// TIA Portal V17 export
// export: Created 2024-08-29T18:23:42.6624587Z, ExportSetting WithDefaults, DisplayName Totally Integrated Automation Portal, DisplayVersion V17 Update 7, DisplayName TIA Portal Openness, DisplayVersion V17 Update 7, DisplayName TIA Portal Version Control Interface, DisplayVersion V17, DisplayName SINAMICS Startdrive Advanced, DisplayVersion V17 SP2, DisplayName SINAMICS Startdrive G110M, G120, G120C, G120D, G120P, G115D, DisplayVersion V17 SP2, DisplayName SINAMICS Startdrive G130, G150, S120, S150, SINAMICS MV, S210, DisplayVersion V17 SP2, DisplayName STEP 7 Professional, DisplayVersion V17 Update 7, DisplayName STEP 7 Safety, DisplayVersion V17 Update 6, DisplayName WinCC Advanced / Unified PC, DisplayVersion V17 Update 7
ORGANIZATION_BLOCK "stationOutputs"   // OB124, LAD, ProgramCycle
TITLE = "Main Program Sweep (Cycle)"
{ S7_Optimized_Access := 'TRUE' }
VERSION : 0.1
// stored: AutoNumber true, IsIECCheckEnabled false, SetENOAutomatically false
   VAR_INPUT
      Initial_Call : Bool;   // Initial call of this OB
      Remanence : Bool;   // =True, if remanent data are available
   END_VAR
   VAR_TEMP
      estopOK : Bool;
   END_VAR
BEGIN

REGION Network 1: PRESENT PARTS
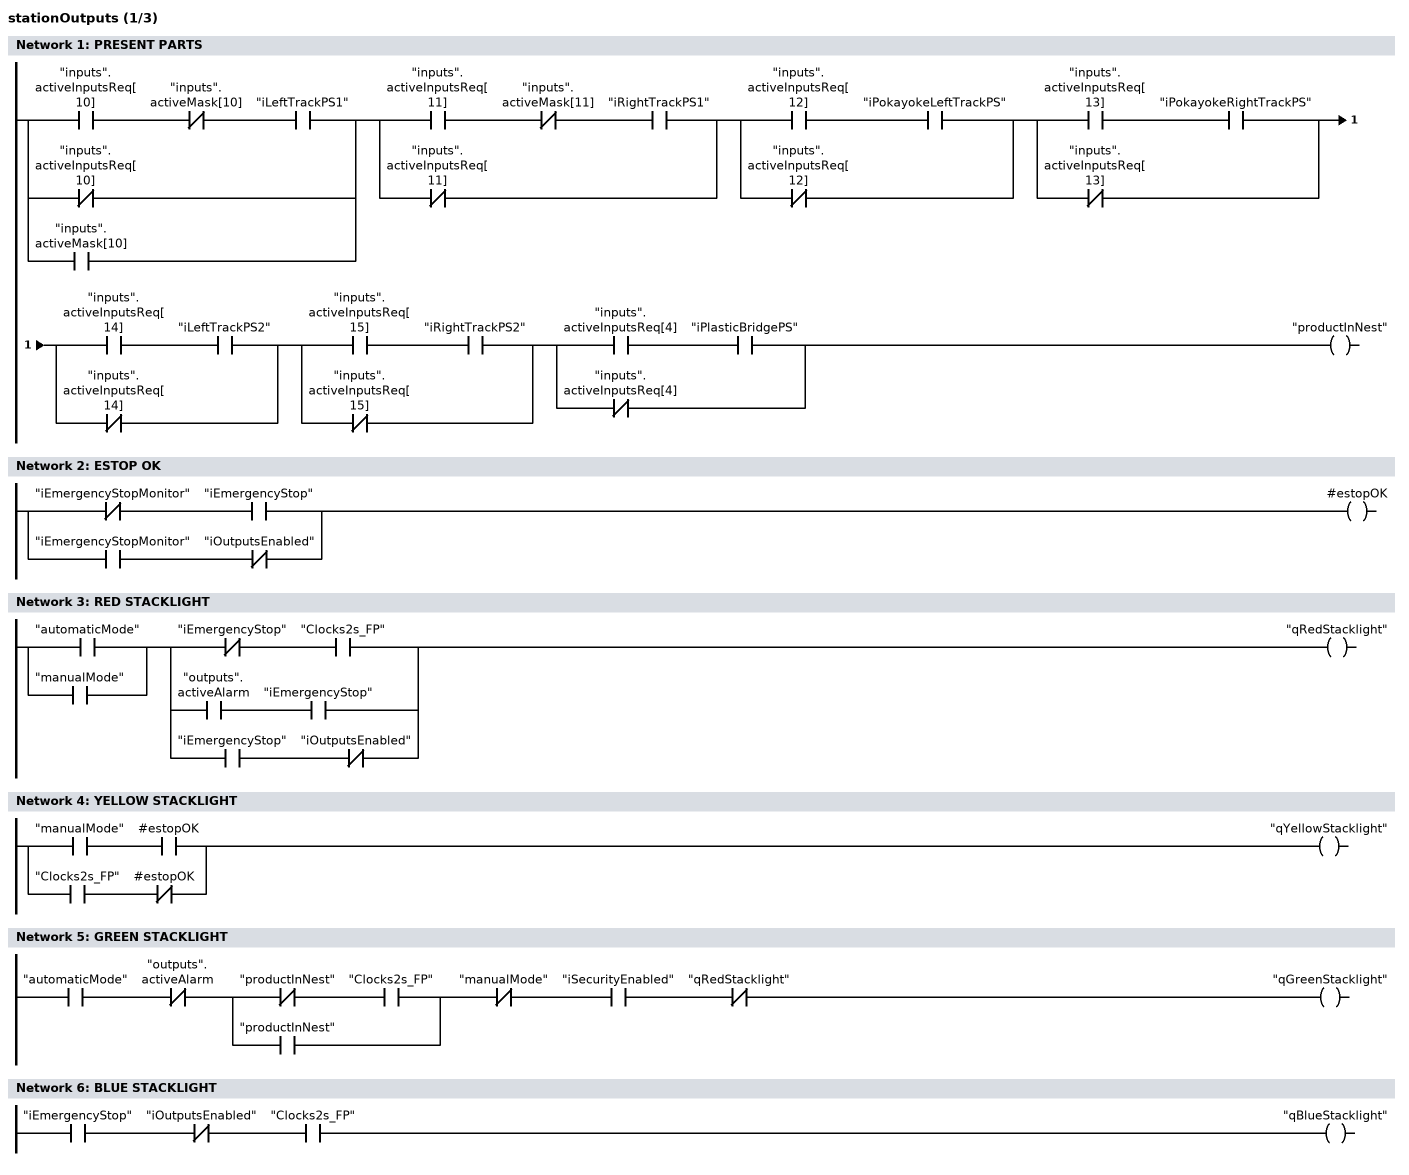
   RUNG wire#powerrail
      Contact( "inputs".activeInputsReq[10] )
      I_Contact( "inputs".activeMask[10] )
      Contact( "iLeftTrackPS1" )
      wire#w1
      Contact( "inputs".activeInputsReq[11] )
      I_Contact( "inputs".activeMask[11] )
      Contact( "iRightTrackPS1" )
      wire#w2
      Contact( "inputs".activeInputsReq[12] )
      Contact( "iPokayokeLeftTrackPS" )
      wire#w3
      Contact( "inputs".activeInputsReq[13] )
      Contact( "iPokayokeRightTrackPS" )
      wire#w4
      Contact( "inputs".activeInputsReq[14] )
      Contact( "iLeftTrackPS2" )
      wire#w5
      Contact( "inputs".activeInputsReq[15] )
      Contact( "iRightTrackPS2" )
      wire#w6
      Contact( "inputs".activeInputsReq[4] )
      Contact( "iPlasticBridgePS" )
      wire#w7
      Coil( "productInNest" )
   END_RUNG
   RUNG wire#powerrail
      I_Contact( "inputs".activeInputsReq[10] )
   END_RUNG wire#w1
   RUNG wire#powerrail
      Contact( "inputs".activeMask[10] )
   END_RUNG wire#w1
   RUNG wire#w1
      I_Contact( "inputs".activeInputsReq[11] )
   END_RUNG wire#w2
   RUNG wire#w2
      I_Contact( "inputs".activeInputsReq[12] )
   END_RUNG wire#w3
   RUNG wire#w3
      I_Contact( "inputs".activeInputsReq[13] )
   END_RUNG wire#w4
   RUNG wire#w4
      I_Contact( "inputs".activeInputsReq[14] )
   END_RUNG wire#w5
   RUNG wire#w5
      I_Contact( "inputs".activeInputsReq[15] )
   END_RUNG wire#w6
   RUNG wire#w6
      I_Contact( "inputs".activeInputsReq[4] )
   END_RUNG wire#w7
   // the same network as SCL:
   "productInNest" := (("inputs".activeInputsReq[10] AND NOT "inputs".activeMask[10] AND "iLeftTrackPS1") OR NOT "inputs".activeInputsReq[10] OR "inputs".activeMask[10]) AND (("inputs".activeInputsReq[11] AND NOT "inputs".activeMask[11] AND "iRightTrackPS1") OR NOT "inputs".activeInputsReq[11]) AND (("inputs".activeInputsReq[12] AND "iPokayokeLeftTrackPS") OR NOT "inputs".activeInputsReq[12]) AND (("inputs".activeInputsReq[13] AND "iPokayokeRightTrackPS") OR NOT "inputs".activeInputsReq[13]) AND (("inputs".activeInputsReq[14] AND "iLeftTrackPS2") OR NOT "inputs".activeInputsReq[14]) AND (("inputs".activeInputsReq[15] AND "iRightTrackPS2") OR NOT "inputs".activeInputsReq[15]) AND (("inputs".activeInputsReq[4] AND "iPlasticBridgePS") OR NOT "inputs".activeInputsReq[4]);
END_REGION

REGION Network 2: ESTOP OK
   RUNG wire#powerrail
      I_Contact( "iEmergencyStopMonitor" )
      Contact( "iEmergencyStop" )
      wire#w1
      Coil( #estopOK )
   END_RUNG
   RUNG wire#powerrail
      Contact( "iEmergencyStopMonitor" )
      I_Contact( "iOutputsEnabled" )
   END_RUNG wire#w1
   // the same network as SCL:
   #estopOK := (NOT "iEmergencyStopMonitor" AND "iEmergencyStop") OR ("iEmergencyStopMonitor" AND NOT "iOutputsEnabled");
END_REGION

REGION Network 3: RED STACKLIGHT
   RUNG wire#powerrail
      Contact( "automaticMode" )
      wire#w1
      I_Contact( "iEmergencyStop" )
      Contact( "Clocks2s_FP" )
      wire#w2
      Coil( "qRedStacklight" )
   END_RUNG
   RUNG wire#powerrail
      Contact( "manualMode" )
   END_RUNG wire#w1
   RUNG wire#w1
      Contact( "outputs".activeAlarm )
      Contact( "iEmergencyStop" )
   END_RUNG wire#w2
   RUNG wire#w1
      Contact( "iEmergencyStop" )
      I_Contact( "iOutputsEnabled" )
   END_RUNG wire#w2
   // the same network as SCL:
   "qRedStacklight" := ("automaticMode" OR "manualMode") AND ((NOT "iEmergencyStop" AND "Clocks2s_FP") OR ("outputs".activeAlarm AND "iEmergencyStop") OR ("iEmergencyStop" AND NOT "iOutputsEnabled"));
END_REGION

REGION Network 4: YELLOW STACKLIGHT
   RUNG wire#powerrail
      Contact( "manualMode" )
      Contact( #estopOK )
      wire#w1
      Coil( "qYellowStacklight" )
   END_RUNG
   RUNG wire#powerrail
      Contact( "Clocks2s_FP" )
      I_Contact( #estopOK )
   END_RUNG wire#w1
   // the same network as SCL:
   "qYellowStacklight" := ("manualMode" AND #estopOK) OR ("Clocks2s_FP" AND NOT #estopOK);
END_REGION

REGION Network 5: GREEN STACKLIGHT
   RUNG wire#powerrail
      Contact( "automaticMode" )
      I_Contact( "outputs".activeAlarm )
      wire#w1
      I_Contact( "productInNest" )
      Contact( "Clocks2s_FP" )
      wire#w2
      I_Contact( "manualMode" )
      Contact( "iSecurityEnabled" )
      I_Contact( "qRedStacklight" )
      Coil( "qGreenStacklight" )
   END_RUNG
   RUNG wire#w1
      Contact( "productInNest" )
   END_RUNG wire#w2
   // the same network as SCL:
   "qGreenStacklight" := "automaticMode" AND NOT "outputs".activeAlarm AND ((NOT "productInNest" AND "Clocks2s_FP") OR "productInNest") AND NOT "manualMode" AND "iSecurityEnabled" AND NOT "qRedStacklight";
END_REGION

REGION Network 6: BLUE STACKLIGHT
   RUNG wire#powerrail
      Contact( "iEmergencyStop" )
      I_Contact( "iOutputsEnabled" )
      Contact( "Clocks2s_FP" )
      Coil( "qBlueStacklight" )
   END_RUNG
   // the same network as SCL:
   "qBlueStacklight" := "iEmergencyStop" AND NOT "iOutputsEnabled" AND "Clocks2s_FP";
END_REGION

REGION Network 7: GREEN INDICATOR
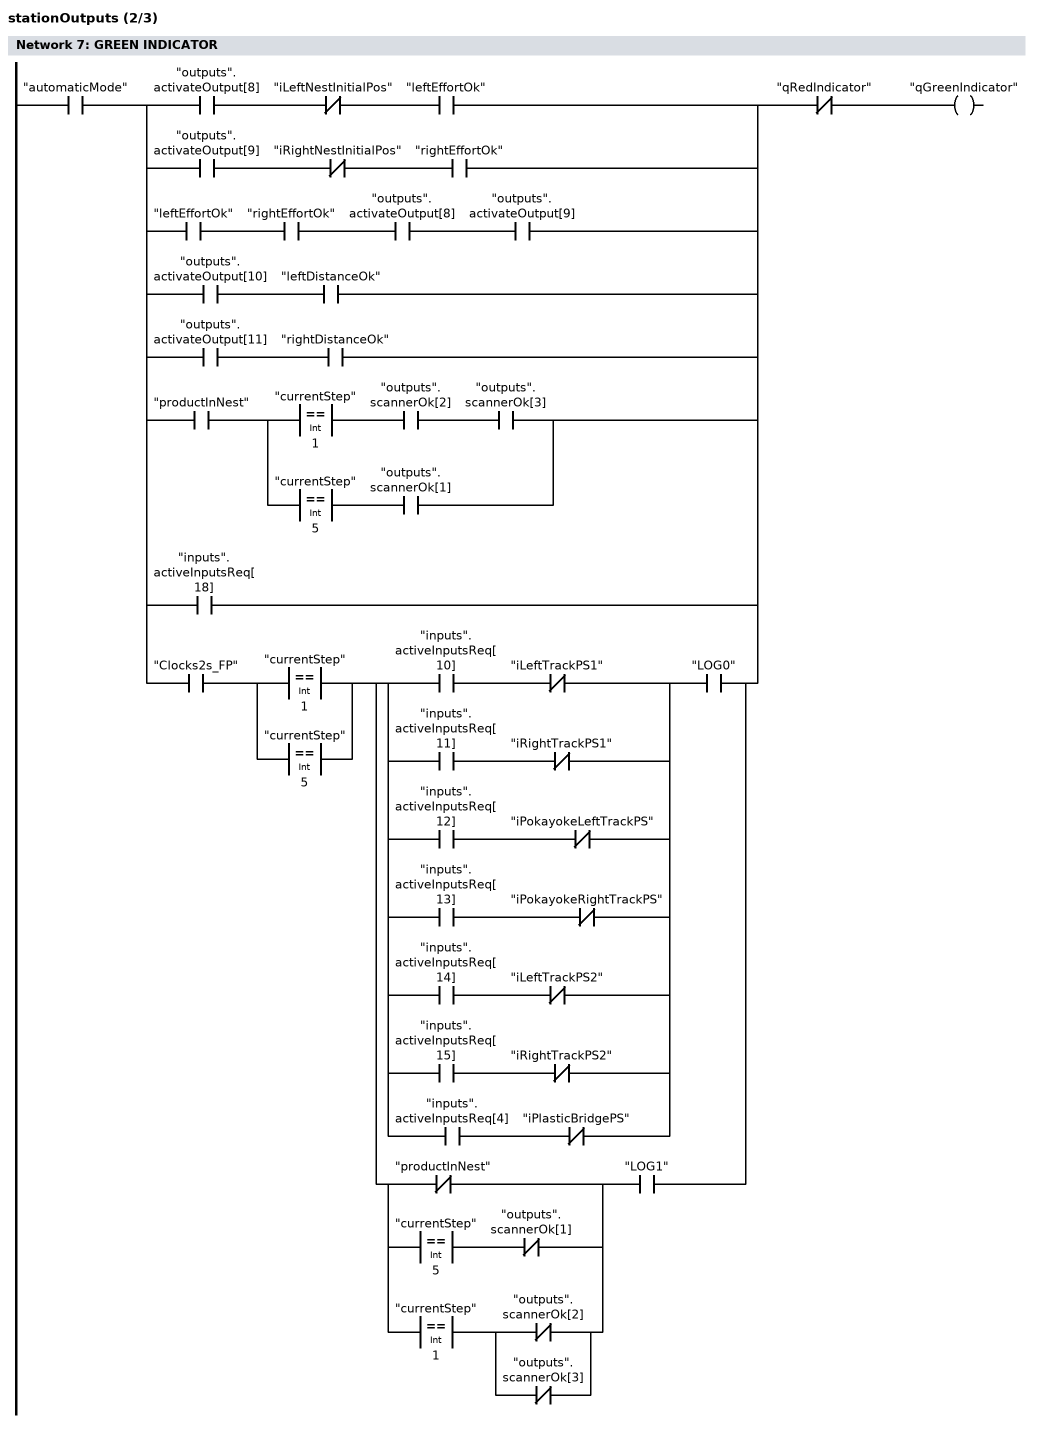
   RUNG wire#powerrail
      Contact( "automaticMode" )
      wire#w1
      Contact( "outputs".activateOutput[8] )
      I_Contact( "iLeftNestInitialPos" )
      Contact( "leftEffortOk" )
      wire#w2
      I_Contact( "qRedIndicator" )
      Coil( "qGreenIndicator" )
   END_RUNG
   RUNG wire#w1
      Contact( "outputs".activateOutput[9] )
      I_Contact( "iRightNestInitialPos" )
      Contact( "rightEffortOk" )
   END_RUNG wire#w2
   RUNG wire#w1
      Contact( "leftEffortOk" )
      Contact( "rightEffortOk" )
      Contact( "outputs".activateOutput[8] )
      Contact( "outputs".activateOutput[9] )
   END_RUNG wire#w2
   RUNG wire#w1
      Contact( "outputs".activateOutput[10] )
      Contact( "leftDistanceOk" )
   END_RUNG wire#w2
   RUNG wire#w1
      Contact( "outputs".activateOutput[11] )
      Contact( "rightDistanceOk" )
   END_RUNG wire#w2
   RUNG wire#w1
      Contact( "productInNest" )
      wire#w3
      { S7_Templates := "SrcType := Int" } EQ_Contact(in1 := "currentStep", in2 := 1)
      Contact( "outputs".scannerOk[2] )
      Contact( "outputs".scannerOk[3] )
   END_RUNG wire#w2
   RUNG wire#w3
      { S7_Templates := "SrcType := Int" } EQ_Contact(in1 := "currentStep", in2 := 5)
      Contact( "outputs".scannerOk[1] )
   END_RUNG wire#w2
   RUNG wire#w1
      Contact( "inputs".activeInputsReq[18] )
   END_RUNG wire#w2
   RUNG wire#w1
      Contact( "Clocks2s_FP" )
      wire#w4
      { S7_Templates := "SrcType := Int" } EQ_Contact(in1 := "currentStep", in2 := 1)
      wire#w5
      Contact( "inputs".activeInputsReq[10] )
      I_Contact( "iLeftTrackPS1" )
      wire#w6
      Contact( "LOG0" )
   END_RUNG wire#w2
   RUNG wire#w4
      { S7_Templates := "SrcType := Int" } EQ_Contact(in1 := "currentStep", in2 := 5)
   END_RUNG wire#w5
   RUNG wire#w5
      Contact( "inputs".activeInputsReq[11] )
      I_Contact( "iRightTrackPS1" )
   END_RUNG wire#w6
   RUNG wire#w5
      Contact( "inputs".activeInputsReq[12] )
      I_Contact( "iPokayokeLeftTrackPS" )
   END_RUNG wire#w6
   RUNG wire#w5
      Contact( "inputs".activeInputsReq[13] )
      I_Contact( "iPokayokeRightTrackPS" )
   END_RUNG wire#w6
   RUNG wire#w5
      Contact( "inputs".activeInputsReq[14] )
      I_Contact( "iLeftTrackPS2" )
   END_RUNG wire#w6
   RUNG wire#w5
      Contact( "inputs".activeInputsReq[15] )
      I_Contact( "iRightTrackPS2" )
   END_RUNG wire#w6
   RUNG wire#w5
      Contact( "inputs".activeInputsReq[4] )
      I_Contact( "iPlasticBridgePS" )
   END_RUNG wire#w6
   RUNG wire#w5
      I_Contact( "productInNest" )
      wire#w7
      Contact( "LOG1" )
   END_RUNG wire#w2
   RUNG wire#w5
      { S7_Templates := "SrcType := Int" } EQ_Contact(in1 := "currentStep", in2 := 5)
      I_Contact( "outputs".scannerOk[1] )
   END_RUNG wire#w7
   RUNG wire#w5
      { S7_Templates := "SrcType := Int" } EQ_Contact(in1 := "currentStep", in2 := 1)
      wire#w8
      I_Contact( "outputs".scannerOk[2] )
   END_RUNG wire#w7
   RUNG wire#w8
      I_Contact( "outputs".scannerOk[3] )
   END_RUNG wire#w7
   // the same network as SCL:
   "qGreenIndicator" := "automaticMode" AND (("outputs".activateOutput[8] AND NOT "iLeftNestInitialPos" AND "leftEffortOk") OR ("outputs".activateOutput[9] AND NOT "iRightNestInitialPos" AND "rightEffortOk") OR ("leftEffortOk" AND "rightEffortOk" AND "outputs".activateOutput[8] AND "outputs".activateOutput[9]) OR ("outputs".activateOutput[10] AND "leftDistanceOk") OR ("outputs".activateOutput[11] AND "rightDistanceOk") OR ("productInNest" AND ((("currentStep" = 1) AND "outputs".scannerOk[2] AND "outputs".scannerOk[3]) OR (("currentStep" = 5) AND "outputs".scannerOk[1]))) OR "inputs".activeInputsReq[18] OR ("Clocks2s_FP" AND (("currentStep" = 1) OR ("currentStep" = 5)) AND (((("inputs".activeInputsReq[10] AND NOT "iLeftTrackPS1") OR ("inputs".activeInputsReq[11] AND NOT "iRightTrackPS1") OR ("inputs".activeInputsReq[12] AND NOT "iPokayokeLeftTrackPS") OR ("inputs".activeInputsReq[13] AND NOT "iPokayokeRightTrackPS") OR ("inputs".activeInputsReq[14] AND NOT "iLeftTrackPS2") OR ("inputs".activeInputsReq[15] AND NOT "iRightTrackPS2") OR ("inputs".activeInputsReq[4] AND NOT "iPlasticBridgePS")) AND "LOG0") OR ((NOT "productInNest" OR (("currentStep" = 5) AND NOT "outputs".scannerOk[1]) OR (("currentStep" = 1) AND (NOT "outputs".scannerOk[2] OR NOT "outputs".scannerOk[3]))) AND "LOG1")))) AND NOT "qRedIndicator";
END_REGION

REGION Network 8: YELLOW INDICATOR
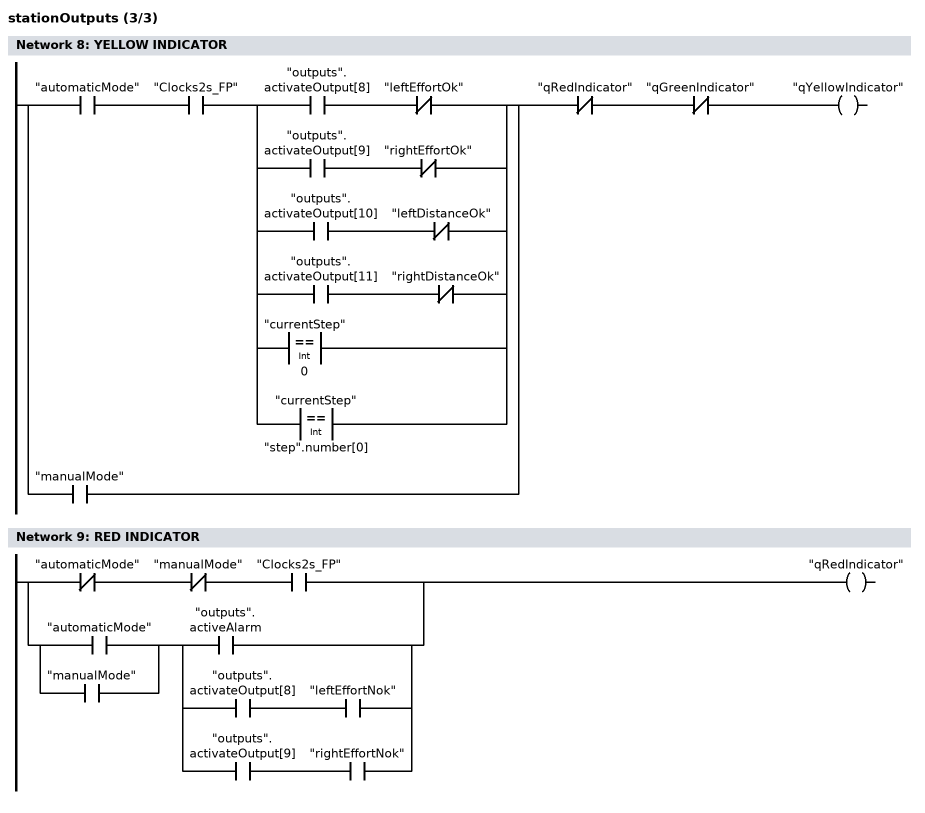
   RUNG wire#powerrail
      Contact( "automaticMode" )
      Contact( "Clocks2s_FP" )
      wire#w1
      Contact( "outputs".activateOutput[8] )
      I_Contact( "leftEffortOk" )
      wire#w2
      I_Contact( "qRedIndicator" )
      I_Contact( "qGreenIndicator" )
      Coil( "qYellowIndicator" )
   END_RUNG
   RUNG wire#w1
      Contact( "outputs".activateOutput[9] )
      I_Contact( "rightEffortOk" )
   END_RUNG wire#w2
   RUNG wire#w1
      Contact( "outputs".activateOutput[10] )
      I_Contact( "leftDistanceOk" )
   END_RUNG wire#w2
   RUNG wire#w1
      Contact( "outputs".activateOutput[11] )
      I_Contact( "rightDistanceOk" )
   END_RUNG wire#w2
   RUNG wire#w1
      { S7_Templates := "SrcType := Int" } EQ_Contact(in1 := "currentStep", in2 := 0)
   END_RUNG wire#w2
   RUNG wire#w1
      { S7_Templates := "SrcType := Int" } EQ_Contact(in1 := "currentStep", in2 := "step".number[0])
   END_RUNG wire#w2
   RUNG wire#powerrail
      Contact( "manualMode" )
   END_RUNG wire#w2
   // the same network as SCL:
   "qYellowIndicator" := (("automaticMode" AND "Clocks2s_FP" AND (("outputs".activateOutput[8] AND NOT "leftEffortOk") OR ("outputs".activateOutput[9] AND NOT "rightEffortOk") OR ("outputs".activateOutput[10] AND NOT "leftDistanceOk") OR ("outputs".activateOutput[11] AND NOT "rightDistanceOk") OR ("currentStep" = 0) OR ("currentStep" = "step".number[0]))) OR "manualMode") AND NOT "qRedIndicator" AND NOT "qGreenIndicator";
END_REGION

REGION Network 9: RED INDICATOR
   RUNG wire#powerrail
      I_Contact( "automaticMode" )
      I_Contact( "manualMode" )
      Contact( "Clocks2s_FP" )
      wire#w1
      Coil( "qRedIndicator" )
   END_RUNG
   RUNG wire#powerrail
      Contact( "automaticMode" )
      wire#w2
      Contact( "outputs".activeAlarm )
   END_RUNG wire#w1
   RUNG wire#powerrail
      Contact( "manualMode" )
   END_RUNG wire#w2
   RUNG wire#w2
      Contact( "outputs".activateOutput[8] )
      Contact( "leftEffortNok" )
   END_RUNG wire#w1
   RUNG wire#w2
      Contact( "outputs".activateOutput[9] )
      Contact( "rightEffortNok" )
   END_RUNG wire#w1
   // the same network as SCL:
   "qRedIndicator" := (NOT "automaticMode" AND NOT "manualMode" AND "Clocks2s_FP") OR (("automaticMode" OR "manualMode") AND ("outputs".activeAlarm OR ("outputs".activateOutput[8] AND "leftEffortNok") OR ("outputs".activateOutput[9] AND "rightEffortNok")));
END_REGION
END_ORGANIZATION_BLOCK
